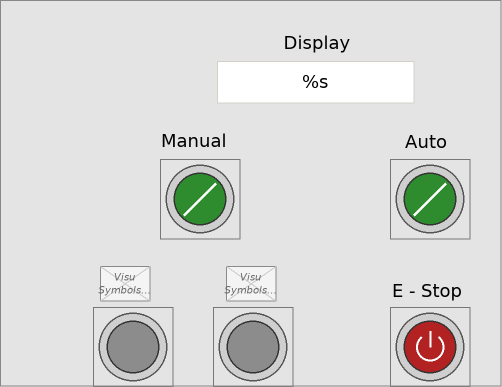
VISUALIZATION HMIControl  // 502x387
    Image (226,266 50x35), image: VisuSymbols.Symbols.ArrowBoldRight
    PushSwitch (88,307 90x80), variable: GVL.qxButtLeft, behaviour: TAP, style: Switch-PushSwitch-Gray
    PushSwitch (208,307 90x80), variable: GVL.qxButtRight, behaviour: TAP, style: Switch-PushSwitch-Gray
    Image (100,266 50x35), image: VisuSymbols.Symbols.ArrowBoldLeft
    Label (119,126 150x30), "Manual"
    RotarySwitch (155,159 90x80), variable: GVL.qxButtManual, behaviour: TOGGLE, style: Switch-RotarySwitch-Green
    RotarySwitch (385,159 90x80), variable: GVL.qxButtAuto, input disabled if: NOT Auto.Home, behaviour: TOGGLE, style: Switch-RotarySwitch-Green
    Label (351,127 150x30), "Auto"
    PowerSwitch (385,307 90x80), variable: GVL.qxButtEmerg, behaviour: TOGGLE, style: Switch-PowerSwitch-Red
    Label (352,276 150x30), "E - Stop"
    Textfield (217,61 197x42), "%s", text variable: TextDisplay.TextDis
    Label (242,28 150x30), "Display"
END_VISUALIZATION

(* stored: Version 1.1.0.1, ProductVersion 3.1.4024.12
   Visu HMIControl: Id {8e0982f4-dcc0-40da-9a15-fb41dd1ecd86} *)
